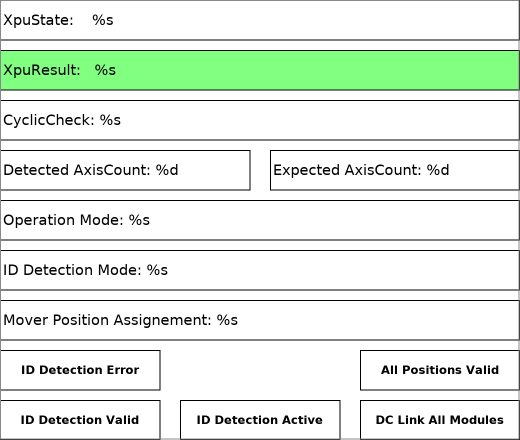
VISUALIZATION XPU_VISU  // 520x440
VAR_IN_OUT
	stXpuState    : ST_XPU_STATE;
  stXpuInfo     : ST_XPU_INFO;
  stXpuStrings  : ST_XPU_STRINGS;
END_VAR
    Rectangle (0,100 520x40), "CyclicCheck: %s", text variable: stXpuStrings.sXpuCyclicCheck
    Rectangle (0,0 520x40), "XpuState: %s", text variable: stXpuStrings.sXpuState
    Rectangle (0,50 520x40), "XpuResult: %s", text variable: stXpuStrings.sXpuResult, colour toggle: (MAIN.eXpuResult = E_PROGRESS.PROGRESS_ERROR)
    Rectangle (360,350 160x40), "All Positions Valid", colour toggle: stXpuInfo.AllPositionsValid
    Rectangle (0,350 160x40), "ID Detection Error", colour toggle: stXpuInfo.IdDetectionError
    Rectangle (0,400 160x40), "ID Detection Valid", colour toggle: stXpuInfo.IdDetectionValid
    Rectangle (180,400 160x40), "ID Detection Active", colour toggle: stXpuInfo.IdDetectionActive
    Rectangle (0,200 520x40), "Operation Mode: %s", text variable: stXpuStrings.sXpuOpMode
    Rectangle (0,250 520x40), "ID Detection Mode: %s", text variable: stXpuStrings.sXpuMoverId_DetectionMode
    Rectangle (0,300 520x40), "Mover Position Assignement: %s", text variable: stXpuStrings.sXpuMoverPosAssignement
    Rectangle (270,150 250x40), "Expected AxisCount: %d", text variable: stXpuInfo.nExpectedAxisCount
    Rectangle (0,150 250x40), "Detected AxisCount: %d", text variable: stXpuInfo.nDetectedAxisCount
    Rectangle (360,400 160x40), "DC Link All Modules", colour toggle: stXpuState.DcLink
END_VISUALIZATION

(* stored: Version 1.1.0.1
   Visu XPU_VISU: Id {bf97327e-e922-4728-90c6-20e9258e2b07} *)
